(* IEC 61131-3 sources: ST_Compiler/, 1 file *)

(* ---- test.st ---- *)
PROGRAM Example
    VAR
        x : INT := 10;
        y : BOOL;
    END_VAR

    y := Add(x, y);  // 函数调用语句

END_PROGRAM
